// TIA Portal V16 export
// export: Created 2021-11-12T13:32:32.9016041Z, ExportSetting WithDefaults, DisplayName Totally Integrated Automation Portal, DisplayVersion V16 Update 3, DisplayName TIA Portal Version Control Interface, DisplayVersion V16 Update 2, DisplayName TIA Portal Openness, DisplayVersion V16 Update 3, DisplayName SINAMICS Startdrive Advanced, DisplayVersion V16 Update 5, DisplayName SINAMICS Startdrive G130, G150, S120, S150, SINAMICS MV, S210, DisplayVersion V16 Update 5, DisplayName SINAMICS Startdrive G110M, G120, G120C, G120D, G120P, G115D, DisplayVersion V16 Update 5, DisplayName STEP 7 Professional, DisplayVersion V16 Update 3, DisplayName STEP 7 Safety, DisplayVersion V16, DisplayName WinCC UA Professional, DisplayVersion V16 Update 3
DATA_BLOCK "HMI_CMD_Zone100"   // DB17
{ S7_Optimized_Access := 'TRUE'; DB_Accessible_From_OPC_UA := 'FALSE' }
VERSION : 0.1
// stored: AutoNumber true, DBAccessibleFromOPCUA false, IsOnlyStoredInLoadMemory false, IsRetainMemResEnabled false, IsWriteProtectedInAS false, MemoryReserve 100
   VAR
      Mode : "UDT_Zone_Command";   // Commands of zone 100
      StationKAS1_Mode { S7_SetPoint := 'True'} : "UDT_Station_Command";   // Commands of station saw KAS1
      StationKAS2_Mode { S7_SetPoint := 'True'} : "UDT_Station_Command";   // Commands of station saw KAS2
      Station110_Mode : "UDT_Station_Command";   // Commands of station 110
      Station120_Mode : "UDT_Station_Command";   // Commands of station 120
      Station1R1_Mode : "UDT_Station_Command";   // Commands of station 1R1
      Station1R2_Mode : "UDT_Station_Command";   // Commands of station 1R2
      Station130_Mode : "UDT_Station_Command";   // Commands of station 130
      Station140_Mode : "UDT_Station_Command";   // Commands of station 140
      Station1R3_Mode : "UDT_Station_Command";   // Commands of station 1R3
      Station1R4_Mode : "UDT_Station_Command";   // Commands of station 1R4
      Station150_Mode : "UDT_Station_Command";   // Commands of station 150
      Station160_Mode : "UDT_Station_Command";   // Commands of station 160
      Station170_Mode : "UDT_Station_Command";   // Commands of station 170
      Station180_Mode : "UDT_Station_Command";   // Commands of station 180
      Station1R5_Mode : "UDT_Station_Command";   // Commands of station 1R5
      Station1R6_Mode : "UDT_Station_Command";   // Commands of station 1R6
      StationBSN1_Mode { S7_SetPoint := 'True'} : "UDT_Station_Command";   // Commands of station furnace BSN1
      StationBSN2_Mode { S7_SetPoint := 'True'} : "UDT_Station_Command";   // Commands of station furnace BSN2
      StationsSum { S7_SetPoint := 'True'} : "UDT_StationsModesCmd";
      xxxxx___Alarms___xxxxx { S7_SetPoint := 'True'} : Byte;
      "UF01-SF01_ES" : "UDT_DI_Mon_Command";   // E-stop 100UF01-SF01
      QQ01_ES { S7_SetPoint := 'True'} : "UDT_DI_Mon_Command";   // E-stop gate 100QQ01
      QQ02_ES { S7_SetPoint := 'True'} : "UDT_DI_Mon_Command";   // E-stop gate 100QQ02
      QQ03_ES { S7_SetPoint := 'True'} : "UDT_DI_Mon_Command";   // E-stop gate 100QQ03
      QQ04_ES { S7_SetPoint := 'True'} : "UDT_DI_Mon_Command";   // E-stop gate 100QQ04
      QQ05_ES { S7_SetPoint := 'True'} : "UDT_DI_Mon_Command";   // E-stop gate 100QQ05
      QQ06_ES { S7_SetPoint := 'True'} : "UDT_DI_Mon_Command";   // E-stop gate 100QQ06
      QQ07_ES { S7_SetPoint := 'True'} : "UDT_DI_Mon_Command";   // E-stop gate 100QQ07
      QQ08_ES { S7_SetPoint := 'True'} : "UDT_DI_Mon_Command";   // E-stop gate 100QQ08
      "RU01-KF01" { S7_SetPoint := 'True'} : "UDT_DI_Mon_Command";   // gate module 100RU01-KF01
      "RU01-KF02" { S7_SetPoint := 'True'} : "UDT_DI_Mon_Command";   // gate module 100RU01-KF01
      "RU01-KF03" { S7_SetPoint := 'True'} : "UDT_DI_Mon_Command";   // gate module 100RU01-KF01
   END_VAR
BEGIN
END_DATA_BLOCK
